{attribute 'linkalways'} 
{attribute 'no_explicit_call' := 'This FB is a CLASS and must be accessed using methods or properties'}
{attribute 'enable_dynamic_creation'}
FUNCTION_BLOCK Collection EXTENDS Disposable IMPLEMENTS I_Collection
VAR
	linkedList : LinkedList;
END_VAR

METHOD PUBLIC AddItem
VAR_INPUT
	Item : ANY;
END_VAR
linkedList.AddLast(Item);
END_METHOD

METHOD PUBLIC Clear
linkedList.Clear();
END_METHOD

METHOD PUBLIC Contains : BOOL;
VAR_INPUT
	Item : ANY;
END_VAR
VAR
	found : I_LinkedListNode;
END_VAR
found := linkedList.Find(Item);
Contains := found <> 0;
END_METHOD

METHOD PUBLIC CopyTo : BOOL
VAR_INPUT
	Destination : ANY;
END_VAR
CopyTo := linkedList.CopyTo(Destination);
END_METHOD

METHOD PUBLIC CopyToLocation : BOOL
VAR_INPUT
	Destination : PVOID;
	DestinationSize : UDINT;
END_VAR
CopyToLocation := linkedList.CopyToLocation(Destination, DestinationSize);
END_METHOD

PROPERTY PUBLIC Count : ULINT
GET
Count := linkedList.Count;
END_GET
END_PROPERTY

METHOD FB_exit : BOOL
VAR_INPUT
	bInCopyCode : BOOL; // if TRUE, the exit method is called for exiting an instance that is copied afterwards (online change).
END_VAR
IF bInCopyCode THEN
	RETURN;
END_IF

Clear();
END_METHOD

METHOD PUBLIC GetEnumerator : I_ForwardEnumerator
GetEnumerator := linkedList.GetEnumerator();
END_METHOD

METHOD RemoveItem : BOOL
VAR_INPUT
	Item : ANY;
END_VAR
RemoveItem := linkedList.RemoveItem(Item);
END_METHOD

END_FUNCTION_BLOCK

(* stored: Version 1.1.0.1, ProductVersion 3.1.4024.12
   POU Collection: Id {065f5ffd-dd59-4040-826f-fb12d2016595}, SpecialFunc None
   Folder Destructor: Id {440fd707-36a1-4231-814c-4260b3a77c94}
   Method AddItem: Id {41518e04-0c64-4bc8-b5d6-07b793d81d8f}
   Method Clear: Id {5a5ff28f-8b9e-4823-a7a9-d8120cde8058}
   Method Contains: Id {240acf57-b71f-4e84-b3f1-497353d5640c}
   Method CopyTo: Id {fc2c1ba9-05c6-4256-9ff8-a81a906f7952}
   Method CopyToLocation: Id {fe6726f8-516e-44c3-aa6e-1b02156054dc}
   Property Count: Id {c1dc2608-40b9-4aa8-ba2d-52b671666be1}
   Get Get: Id {4254f1fb-bbf3-4a13-a860-009d211704df}
   Method FB_exit: Id {07774179-de13-4358-99c3-6233681d2bad}
   Method GetEnumerator: Id {3a50b611-1a11-468e-980e-9b675fd835e6}
   Method RemoveItem: Id {6fc8d20b-52fd-455f-9293-68105648121c} *)
